LIN {X -19.393, Y 137.224, Z 298.25, A 0, B 90, C 0, E1 0, E2 0, E3 0, E4 0} C_DIS
LIN {X -14.94, Y 135.645, Z 298.25, A 0, B 90, C 0, E1 0, E2 0, E3 0, E4 0} C_DIS
LIN {X -10.792, Y 133.376, Z 298.25, A 0, B 90, C 0, E1 0, E2 0, E3 0, E4 0} C_DIS
LIN {X -6.941, Y 130.631, Z 298.25, A 0, B 90, C 0, E1 0, E2 0, E3 0, E4 0} C_DIS
LIN {X -3.341, Y 127.563, Z 298.25, A 0, B 90, C 0, E1 0, E2 0, E3 0, E4 0} C_DIS
LIN {X 0, Y 124.352, Z 298.25, A 0, B 90, C 0, E1 0, E2 0, E3 0, E4 0} C_DIS
LIN {X 3.004, Y 120.935, Z 298.25, A 0, B 90, C 0, E1 0, E2 0, E3 0, E4 0} C_DIS
LIN {X 6.227, Y 117.473, Z 298.25, A 0, B 90, C 0, E1 0, E2 0, E3 0, E4 0} C_DIS
LIN {X 9.503, Y 114.059, Z 298.25, A 0, B 90, C 0, E1 0, E2 0, E3 0, E4 0} C_DIS
LIN {X 12.968, Y 110.84, Z 298.25, A 0, B 90, C 0, E1 0, E2 0, E3 0, E4 0} C_DIS
LIN {X 16.832, Y 108.123, Z 298.25, A 0, B 90, C 0, E1 0, E2 0, E3 0, E4 0} C_DIS
LIN {X 21.253, Y 106.495, Z 298.25, A 0, B 90, C 0, E1 0, E2 0, E3 0, E4 0} C_DIS
LIN {X 25.964, Y 106.394, Z 298.25, A 0, B 90, C 0, E1 0, E2 0, E3 0, E4 0} C_DIS
LIN {X 30.572, Y 107.44, Z 298.25, A 0, B 90, C 0, E1 0, E2 0, E3 0, E4 0} C_DIS
LIN {X 35.02, Y 109.05, Z 298.25, A 0, B 90, C 0, E1 0, E2 0, E3 0, E4 0} C_DIS
LIN {X 39.382, Y 110.883, Z 298.25, A 0, B 90, C 0, E1 0, E2 0, E3 0, E4 0} C_DIS
LIN {X 43.728, Y 112.754, Z 298.25, A 0, B 90, C 0, E1 0, E2 0, E3 0, E4 0} C_DIS
LIN {X 48.108, Y 114.542, Z 298.25, A 0, B 90, C 0, E1 0, E2 0, E3 0, E4 0} C_DIS
LIN {X 52.558, Y 116.148, Z 298.25, A 0, B 90, C 0, E1 0, E2 0, E3 0, E4 0} C_DIS
LIN {X 57.101, Y 117.467, Z 298.25, A 0, B 90, C 0, E1 0, E2 0, E3 0, E4 0} C_DIS
LIN {X 61.743, Y 118.371, Z 298.25, A 0, B 90, C 0, E1 0, E2 0, E3 0, E4 0} C_DIS
LIN {X 66.459, Y 118.689, Z 298.25, A 0, B 90, C 0, E1 0, E2 0, E3 0, E4 0} C_DIS
LIN {X 71.159, Y 118.207, Z 298.25, A 0, B 90, C 0, E1 0, E2 0, E3 0, E4 0} C_DIS
LIN {X 75.634, Y 116.707, Z 298.25, A 0, B 90, C 0, E1 0, E2 0, E3 0, E4 0} C_DIS
LIN {X 79.57, Y 114.108, Z 298.25, A 0, B 90, C 0, E1 0, E2 0, E3 0, E4 0} C_DIS
LIN {X 82.708, Y 110.582, Z 298.25, A 0, B 90, C 0, E1 0, E2 0, E3 0, E4 0} C_DIS
LIN {X 84.997, Y 106.45, Z 298.25, A 0, B 90, C 0, E1 0, E2 0, E3 0, E4 0} C_DIS
LIN {X 86.553, Y 101.986, Z 298.25, A 0, B 90, C 0, E1 0, E2 0, E3 0, E4 0} C_DIS
LIN {X 87.536, Y 97.36, Z 298.25, A 0, B 90, C 0, E1 0, E2 0, E3 0, E4 0} C_DIS
LIN {X 88.091, Y 92.663, Z 298.25, A 0, B 90, C 0, E1 0, E2 0, E3 0, E4 0} C_DIS
LIN {X 88.341, Y 87.938, Z 298.25, A 0, B 90, C 0, E1 0, E2 0, E3 0, E4 0} C_DIS
LIN {X 88.398, Y 83.207, Z 298.25, A 0, B 90, C 0, E1 0, E2 0, E3 0, E4 0} C_DIS
LIN {X 88.377, Y 78.476, Z 298.25, A 0, B 90, C 0, E1 0, E2 0, E3 0, E4 0} C_DIS
LIN {X 88.427, Y 73.745, Z 298.25, A 0, B 90, C 0, E1 0, E2 0, E3 0, E4 0} C_DIS
LIN {X 88.78, Y 69.029, Z 298.25, A 0, B 90, C 0, E1 0, E2 0, E3 0, E4 0} C_DIS
LIN {X 89.835, Y 64.425, Z 298.25, A 0, B 90, C 0, E1 0, E2 0, E3 0, E4 0} C_DIS
LIN {X 92.094, Y 60.292, Z 298.25, A 0, B 90, C 0, E1 0, E2 0, E3 0, E4 0} C_DIS
LIN {X 95.553, Y 57.088, Z 298.25, A 0, B 90, C 0, E1 0, E2 0, E3 0, E4 0} C_DIS
LIN {X 99.64, Y 54.714, Z 298.25, A 0, B 90, C 0, E1 0, E2 0, E3 0, E4 0} C_DIS
LIN {X 103.963, Y 52.792, Z 298.25, A 0, B 90, C 0, E1 0, E2 0, E3 0, E4 0} C_DIS
LIN {X 108.359, Y 51.043, Z 298.25, A 0, B 90, C 0, E1 0, E2 0, E3 0, E4 0} C_DIS
LIN {X 112.757, Y 49.297, Z 298.25, A 0, B 90, C 0, E1 0, E2 0, E3 0, E4 0} C_DIS
LIN {X 117.106, Y 47.436, Z 298.25, A 0, B 90, C 0, E1 0, E2 0, E3 0, E4 0} C_DIS
LIN {X 121.359, Y 45.364, Z 298.25, A 0, B 90, C 0, E1 0, E2 0, E3 0, E4 0} C_DIS
LIN {X 125.45, Y 42.989, Z 298.25, A 0, B 90, C 0, E1 0, E2 0, E3 0, E4 0} C_DIS
LIN {X 129.281, Y 40.217, Z 298.25, A 0, B 90, C 0, E1 0, E2 0, E3 0, E4 0} C_DIS
LIN {X 132.696, Y 36.95, Z 298.25, A 0, B 90, C 0, E1 0, E2 0, E3 0, E4 0} C_DIS
LIN {X 135.457, Y 33.118, Z 298.25, A 0, B 90, C 0, E1 0, E2 0, E3 0, E4 0} C_DIS
LIN {X 137.252, Y 28.754, Z 298.25, A 0, B 90, C 0, E1 0, E2 0, E3 0, E4 0} C_DIS
LIN {X 137.838, Y 24.073, Z 298.25, A 0, B 90, C 0, E1 0, E2 0, E3 0, E4 0} C_DIS
LIN {X 137.224, Y 19.393, Z 298.25, A 0, B 90, C 0, E1 0, E2 0, E3 0, E4 0} C_DIS
LIN {X 135.645, Y 14.94, Z 298.25, A 0, B 90, C 0, E1 0, E2 0, E3 0, E4 0} C_DIS
LIN {X 133.376, Y 10.792, Z 298.25, A 0, B 90, C 0, E1 0, E2 0, E3 0, E4 0} C_DIS
LIN {X 130.631, Y 6.941, Z 298.25, A 0, B 90, C 0, E1 0, E2 0, E3 0, E4 0} C_DIS
LIN {X 127.563, Y 3.341, Z 298.25, A 0, B 90, C 0, E1 0, E2 0, E3 0, E4 0} C_DIS
LIN {X 124.352, Y 0, Z 298.25, A 0, B 90, C 0, E1 0, E2 0, E3 0, E4 0} C_DIS
LIN {X 120.935, Y -3.004, Z 298.25, A 0, B 90, C 0, E1 0, E2 0, E3 0, E4 0} C_DIS
LIN {X 117.473, Y -6.227, Z 298.25, A 0, B 90, C 0, E1 0, E2 0, E3 0, E4 0} C_DIS
LIN {X 114.059, Y -9.503, Z 298.25, A 0, B 90, C 0, E1 0, E2 0, E3 0, E4 0} C_DIS
LIN {X 110.84, Y -12.968, Z 298.25, A 0, B 90, C 0, E1 0, E2 0, E3 0, E4 0} C_DIS
LIN {X 108.123, Y -16.832, Z 298.25, A 0, B 90, C 0, E1 0, E2 0, E3 0, E4 0} C_DIS
LIN {X 106.495, Y -21.253, Z 298.25, A 0, B 90, C 0, E1 0, E2 0, E3 0, E4 0} C_DIS
LIN {X 106.394, Y -25.964, Z 298.25, A 0, B 90, C 0, E1 0, E2 0, E3 0, E4 0} C_DIS
LIN {X 107.44, Y -30.572, Z 298.25, A 0, B 90, C 0, E1 0, E2 0, E3 0, E4 0} C_DIS
LIN {X 109.05, Y -35.02, Z 298.25, A 0, B 90, C 0, E1 0, E2 0, E3 0, E4 0} C_DIS
LIN {X 110.883, Y -39.382, Z 298.25, A 0, B 90, C 0, E1 0, E2 0, E3 0, E4 0} C_DIS
LIN {X 112.754, Y -43.728, Z 298.25, A 0, B 90, C 0, E1 0, E2 0, E3 0, E4 0} C_DIS
LIN {X 114.542, Y -48.108, Z 298.25, A 0, B 90, C 0, E1 0, E2 0, E3 0, E4 0} C_DIS
LIN {X 116.148, Y -52.558, Z 298.25, A 0, B 90, C 0, E1 0, E2 0, E3 0, E4 0} C_DIS
LIN {X 117.467, Y -57.101, Z 298.25, A 0, B 90, C 0, E1 0, E2 0, E3 0, E4 0} C_DIS
LIN {X 118.371, Y -61.743, Z 298.25, A 0, B 90, C 0, E1 0, E2 0, E3 0, E4 0} C_DIS
LIN {X 118.689, Y -66.459, Z 298.25, A 0, B 90, C 0, E1 0, E2 0, E3 0, E4 0} C_DIS
LIN {X 118.207, Y -71.159, Z 298.25, A 0, B 90, C 0, E1 0, E2 0, E3 0, E4 0} C_DIS
LIN {X 116.707, Y -75.634, Z 298.25, A 0, B 90, C 0, E1 0, E2 0, E3 0, E4 0} C_DIS
LIN {X 114.108, Y -79.57, Z 298.25, A 0, B 90, C 0, E1 0, E2 0, E3 0, E4 0} C_DIS
LIN {X 110.582, Y -82.708, Z 298.25, A 0, B 90, C 0, E1 0, E2 0, E3 0, E4 0} C_DIS
LIN {X 106.45, Y -84.997, Z 298.25, A 0, B 90, C 0, E1 0, E2 0, E3 0, E4 0} C_DIS
LIN {X 101.986, Y -86.553, Z 298.25, A 0, B 90, C 0, E1 0, E2 0, E3 0, E4 0} C_DIS
LIN {X 97.36, Y -87.536, Z 298.25, A 0, B 90, C 0, E1 0, E2 0, E3 0, E4 0} C_DIS
LIN {X 92.663, Y -88.091, Z 298.25, A 0, B 90, C 0, E1 0, E2 0, E3 0, E4 0} C_DIS
LIN {X 87.938, Y -88.341, Z 298.25, A 0, B 90, C 0, E1 0, E2 0, E3 0, E4 0} C_DIS
LIN {X 83.207, Y -88.398, Z 298.25, A 0, B 90, C 0, E1 0, E2 0, E3 0, E4 0} C_DIS
LIN {X 78.476, Y -88.377, Z 298.25, A 0, B 90, C 0, E1 0, E2 0, E3 0, E4 0} C_DIS
LIN {X 73.745, Y -88.427, Z 298.25, A 0, B 90, C 0, E1 0, E2 0, E3 0, E4 0} C_DIS
LIN {X 69.029, Y -88.78, Z 298.25, A 0, B 90, C 0, E1 0, E2 0, E3 0, E4 0} C_DIS
LIN {X 64.425, Y -89.835, Z 298.25, A 0, B 90, C 0, E1 0, E2 0, E3 0, E4 0} C_DIS
LIN {X 60.292, Y -92.094, Z 298.25, A 0, B 90, C 0, E1 0, E2 0, E3 0, E4 0} C_DIS
LIN {X 57.088, Y -95.553, Z 298.25, A 0, B 90, C 0, E1 0, E2 0, E3 0, E4 0} C_DIS
LIN {X 54.714, Y -99.64, Z 298.25, A 0, B 90, C 0, E1 0, E2 0, E3 0, E4 0} C_DIS
LIN {X 52.792, Y -103.963, Z 298.25, A 0, B 90, C 0, E1 0, E2 0, E3 0, E4 0} C_DIS
LIN {X 51.043, Y -108.359, Z 298.25, A 0, B 90, C 0, E1 0, E2 0, E3 0, E4 0} C_DIS
LIN {X 49.297, Y -112.757, Z 298.25, A 0, B 90, C 0, E1 0, E2 0, E3 0, E4 0} C_DIS
LIN {X 47.436, Y -117.106, Z 298.25, A 0, B 90, C 0, E1 0, E2 0, E3 0, E4 0} C_DIS
LIN {X 45.364, Y -121.359, Z 298.25, A 0, B 90, C 0, E1 0, E2 0, E3 0, E4 0} C_DIS
LIN {X 42.989, Y -125.45, Z 298.25, A 0, B 90, C 0, E1 0, E2 0, E3 0, E4 0} C_DIS
LIN {X 40.217, Y -129.281, Z 298.25, A 0, B 90, C 0, E1 0, E2 0, E3 0, E4 0} C_DIS
LIN {X 36.95, Y -132.696, Z 298.25, A 0, B 90, C 0, E1 0, E2 0, E3 0, E4 0} C_DIS
LIN {X 33.118, Y -135.457, Z 298.25, A 0, B 90, C 0, E1 0, E2 0, E3 0, E4 0} C_DIS
LIN {X 28.754, Y -137.252, Z 298.25, A 0, B 90, C 0, E1 0, E2 0, E3 0, E4 0} C_DIS
LIN {X 24.073, Y -137.838, Z 298.25, A 0, B 90, C 0, E1 0, E2 0, E3 0, E4 0} C_DIS
LIN {X 19.393, Y -137.224, Z 298.25, A 0, B 90, C 0, E1 0, E2 0, E3 0, E4 0} C_DIS
LIN {X 14.94, Y -135.645, Z 298.25, A 0, B 90, C 0, E1 0, E2 0, E3 0, E4 0} C_DIS
LIN {X 10.792, Y -133.376, Z 298.25, A 0, B 90, C 0, E1 0, E2 0, E3 0, E4 0} C_DIS
LIN {X 6.941, Y -130.631, Z 298.25, A 0, B 90, C 0, E1 0, E2 0, E3 0, E4 0} C_DIS
LIN {X 3.341, Y -127.563, Z 298.25, A 0, B 90, C 0, E1 0, E2 0, E3 0, E4 0} C_DIS
LIN {X 0, Y -124.352, Z 298.25, A 0, B 90, C 0, E1 0, E2 0, E3 0, E4 0} C_DIS
LIN {X -3.004, Y -120.935, Z 298.25, A 0, B 90, C 0, E1 0, E2 0, E3 0, E4 0} C_DIS
LIN {X -6.227, Y -117.473, Z 298.25, A 0, B 90, C 0, E1 0, E2 0, E3 0, E4 0} C_DIS
LIN {X -9.503, Y -114.059, Z 298.25, A 0, B 90, C 0, E1 0, E2 0, E3 0, E4 0} C_DIS
LIN {X -12.968, Y -110.84, Z 298.25, A 0, B 90, C 0, E1 0, E2 0, E3 0, E4 0} C_DIS
LIN {X -16.832, Y -108.123, Z 298.25, A 0, B 90, C 0, E1 0, E2 0, E3 0, E4 0} C_DIS
LIN {X -21.253, Y -106.495, Z 298.25, A 0, B 90, C 0, E1 0, E2 0, E3 0, E4 0} C_DIS
LIN {X -25.964, Y -106.394, Z 298.25, A 0, B 90, C 0, E1 0, E2 0, E3 0, E4 0} C_DIS
LIN {X -30.572, Y -107.44, Z 298.25, A 0, B 90, C 0, E1 0, E2 0, E3 0, E4 0} C_DIS
LIN {X -35.02, Y -109.05, Z 298.25, A 0, B 90, C 0, E1 0, E2 0, E3 0, E4 0} C_DIS
LIN {X -39.382, Y -110.883, Z 298.25, A 0, B 90, C 0, E1 0, E2 0, E3 0, E4 0} C_DIS
LIN {X -43.728, Y -112.754, Z 298.25, A 0, B 90, C 0, E1 0, E2 0, E3 0, E4 0} C_DIS
LIN {X -48.108, Y -114.542, Z 298.25, A 0, B 90, C 0, E1 0, E2 0, E3 0, E4 0} C_DIS
LIN {X -52.558, Y -116.148, Z 298.25, A 0, B 90, C 0, E1 0, E2 0, E3 0, E4 0} C_DIS
LIN {X -57.101, Y -117.467, Z 298.25, A 0, B 90, C 0, E1 0, E2 0, E3 0, E4 0} C_DIS
LIN {X -61.743, Y -118.371, Z 298.25, A 0, B 90, C 0, E1 0, E2 0, E3 0, E4 0} C_DIS
LIN {X -66.459, Y -118.689, Z 298.25, A 0, B 90, C 0, E1 0, E2 0, E3 0, E4 0} C_DIS
LIN {X -71.159, Y -118.207, Z 298.25, A 0, B 90, C 0, E1 0, E2 0, E3 0, E4 0} C_DIS
LIN {X -75.634, Y -116.707, Z 298.25, A 0, B 90, C 0, E1 0, E2 0, E3 0, E4 0} C_DIS
LIN {X -79.57, Y -114.108, Z 298.25, A 0, B 90, C 0, E1 0, E2 0, E3 0, E4 0} C_DIS
LIN {X -82.708, Y -110.582, Z 298.25, A 0, B 90, C 0, E1 0, E2 0, E3 0, E4 0} C_DIS
LIN {X -84.997, Y -106.45, Z 298.25, A 0, B 90, C 0, E1 0, E2 0, E3 0, E4 0} C_DIS
LIN {X -86.553, Y -101.986, Z 298.25, A 0, B 90, C 0, E1 0, E2 0, E3 0, E4 0} C_DIS
LIN {X -87.536, Y -97.36, Z 298.25, A 0, B 90, C 0, E1 0, E2 0, E3 0, E4 0} C_DIS
LIN {X -88.091, Y -92.663, Z 298.25, A 0, B 90, C 0, E1 0, E2 0, E3 0, E4 0} C_DIS
LIN {X -88.341, Y -87.938, Z 298.25, A 0, B 90, C 0, E1 0, E2 0, E3 0, E4 0} C_DIS
LIN {X -88.398, Y -83.207, Z 298.25, A 0, B 90, C 0, E1 0, E2 0, E3 0, E4 0} C_DIS
LIN {X -88.377, Y -78.476, Z 298.25, A 0, B 90, C 0, E1 0, E2 0, E3 0, E4 0} C_DIS
LIN {X -88.427, Y -73.745, Z 298.25, A 0, B 90, C 0, E1 0, E2 0, E3 0, E4 0} C_DIS
LIN {X -88.78, Y -69.029, Z 298.25, A 0, B 90, C 0, E1 0, E2 0, E3 0, E4 0} C_DIS
LIN {X -89.835, Y -64.425, Z 298.25, A 0, B 90, C 0, E1 0, E2 0, E3 0, E4 0} C_DIS
LIN {X -92.094, Y -60.292, Z 298.25, A 0, B 90, C 0, E1 0, E2 0, E3 0, E4 0} C_DIS
LIN {X -95.553, Y -57.088, Z 298.25, A 0, B 90, C 0, E1 0, E2 0, E3 0, E4 0} C_DIS
LIN {X -99.64, Y -54.714, Z 298.25, A 0, B 90, C 0, E1 0, E2 0, E3 0, E4 0} C_DIS
LIN {X -103.963, Y -52.792, Z 298.25, A 0, B 90, C 0, E1 0, E2 0, E3 0, E4 0} C_DIS
LIN {X -108.359, Y -51.043, Z 298.25, A 0, B 90, C 0, E1 0, E2 0, E3 0, E4 0} C_DIS
LIN {X -112.757, Y -49.297, Z 298.25, A 0, B 90, C 0, E1 0, E2 0, E3 0, E4 0} C_DIS
LIN {X -117.106, Y -47.436, Z 298.25, A 0, B 90, C 0, E1 0, E2 0, E3 0, E4 0} C_DIS
LIN {X -121.359, Y -45.364, Z 298.25, A 0, B 90, C 0, E1 0, E2 0, E3 0, E4 0} C_DIS
LIN {X -125.45, Y -42.989, Z 298.25, A 0, B 90, C 0, E1 0, E2 0, E3 0, E4 0} C_DIS
LIN {X -129.281, Y -40.217, Z 298.25, A 0, B 90, C 0, E1 0, E2 0, E3 0, E4 0} C_DIS
LIN {X -132.696, Y -36.95, Z 298.25, A 0, B 90, C 0, E1 0, E2 0, E3 0, E4 0} C_DIS
LIN {X -135.457, Y -33.118, Z 298.25, A 0, B 90, C 0, E1 0, E2 0, E3 0, E4 0} C_DIS
LIN {X -137.252, Y -28.754, Z 298.25, A 0, B 90, C 0, E1 0, E2 0, E3 0, E4 0} C_DIS
LIN {X -137.838, Y -24.073, Z 298.25, A 0, B 90, C 0, E1 0, E2 0, E3 0, E4 0} C_DIS
LIN {X -137.224, Y -19.393, Z 298.25, A 0, B 90, C 0, E1 0, E2 0, E3 0, E4 0} C_DIS
LIN {X -135.645, Y -14.94, Z 298.25, A 0, B 90, C 0, E1 0, E2 0, E3 0, E4 0} C_DIS
LIN {X -133.376, Y -10.792, Z 298.25, A 0, B 90, C 0, E1 0, E2 0, E3 0, E4 0} C_DIS
LIN {X -130.631, Y -6.941, Z 298.25, A 0, B 90, C 0, E1 0, E2 0, E3 0, E4 0} C_DIS
LIN {X -127.563, Y -3.341, Z 298.25, A 0, B 90, C 0, E1 0, E2 0, E3 0, E4 0} C_DIS
LIN {X -125.319, Y 0, Z 300.75, A 0, B 90, C 0, E1 0, E2 0, E3 0, E4 0} C_DIS
LIN {X -121.855, Y 3.043, Z 300.75, A 0, B 90, C 0, E1 0, E2 0, E3 0, E4 0} C_DIS
LIN {X -118.342, Y 6.3, Z 300.75, A 0, B 90, C 0, E1 0, E2 0, E3 0, E4 0} C_DIS
LIN {X -114.881, Y 9.612, Z 300.75, A 0, B 90, C 0, E1 0, E2 0, E3 0, E4 0} C_DIS
LIN {X -111.625, Y 13.124, Z 300.75, A 0, B 90, C 0, E1 0, E2 0, E3 0, E4 0} C_DIS
LIN {X -108.897, Y 17.052, Z 300.75, A 0, B 90, C 0, E1 0, E2 0, E3 0, E4 0} C_DIS
LIN {X -107.308, Y 21.549, Z 300.75, A 0, B 90, C 0, E1 0, E2 0, E3 0, E4 0} C_DIS
LIN {X -107.291, Y 26.32, Z 300.75, A 0, B 90, C 0, E1 0, E2 0, E3 0, E4 0} C_DIS
LIN {X -108.43, Y 30.967, Z 300.75, A 0, B 90, C 0, E1 0, E2 0, E3 0, E4 0} C_DIS
LIN {X -110.13, Y 35.445, Z 300.75, A 0, B 90, C 0, E1 0, E2 0, E3 0, E4 0} C_DIS
LIN {X -112.047, Y 39.836, Z 300.75, A 0, B 90, C 0, E1 0, E2 0, E3 0, E4 0} C_DIS
LIN {X -113.995, Y 44.212, Z 300.75, A 0, B 90, C 0, E1 0, E2 0, E3 0, E4 0} C_DIS
LIN {X -115.852, Y 48.629, Z 300.75, A 0, B 90, C 0, E1 0, E2 0, E3 0, E4 0} C_DIS
LIN {X -117.516, Y 53.121, Z 300.75, A 0, B 90, C 0, E1 0, E2 0, E3 0, E4 0} C_DIS
LIN {X -118.876, Y 57.713, Z 300.75, A 0, B 90, C 0, E1 0, E2 0, E3 0, E4 0} C_DIS
LIN {X -119.801, Y 62.411, Z 300.75, A 0, B 90, C 0, E1 0, E2 0, E3 0, E4 0} C_DIS
LIN {X -120.113, Y 67.188, Z 300.75, A 0, B 90, C 0, E1 0, E2 0, E3 0, E4 0} C_DIS
LIN {X -119.591, Y 71.942, Z 300.75, A 0, B 90, C 0, E1 0, E2 0, E3 0, E4 0} C_DIS
LIN {X -118.014, Y 76.452, Z 300.75, A 0, B 90, C 0, E1 0, E2 0, E3 0, E4 0} C_DIS
LIN {X -115.31, Y 80.389, Z 300.75, A 0, B 90, C 0, E1 0, E2 0, E3 0, E4 0} C_DIS
LIN {X -111.675, Y 83.492, Z 300.75, A 0, B 90, C 0, E1 0, E2 0, E3 0, E4 0} C_DIS
LIN {X -107.444, Y 85.723, Z 300.75, A 0, B 90, C 0, E1 0, E2 0, E3 0, E4 0} C_DIS
LIN {X -102.895, Y 87.212, Z 300.75, A 0, B 90, C 0, E1 0, E2 0, E3 0, E4 0} C_DIS
LIN {X -98.194, Y 88.123, Z 300.75, A 0, B 90, C 0, E1 0, E2 0, E3 0, E4 0} C_DIS
LIN {X -93.428, Y 88.603, Z 300.75, A 0, B 90, C 0, E1 0, E2 0, E3 0, E4 0} C_DIS
LIN {X -88.641, Y 88.778, Z 300.75, A 0, B 90, C 0, E1 0, E2 0, E3 0, E4 0} C_DIS
LIN {X -83.851, Y 88.757, Z 300.75, A 0, B 90, C 0, E1 0, E2 0, E3 0, E4 0} C_DIS
LIN {X -79.061, Y 88.659, Z 300.75, A 0, B 90, C 0, E1 0, E2 0, E3 0, E4 0} C_DIS
LIN {X -74.27, Y 88.63, Z 300.75, A 0, B 90, C 0, E1 0, E2 0, E3 0, E4 0} C_DIS
LIN {X -69.489, Y 88.903, Z 300.75, A 0, B 90, C 0, E1 0, E2 0, E3 0, E4 0} C_DIS
LIN {X -64.808, Y 89.881, Z 300.75, A 0, B 90, C 0, E1 0, E2 0, E3 0, E4 0} C_DIS
LIN {X -60.582, Y 92.09, Z 300.75, A 0, B 90, C 0, E1 0, E2 0, E3 0, E4 0} C_DIS
LIN {X -57.303, Y 95.559, Z 300.75, A 0, B 90, C 0, E1 0, E2 0, E3 0, E4 0} C_DIS
LIN {X -54.9, Y 99.697, Z 300.75, A 0, B 90, C 0, E1 0, E2 0, E3 0, E4 0} C_DIS
LIN {X -52.978, Y 104.085, Z 300.75, A 0, B 90, C 0, E1 0, E2 0, E3 0, E4 0} C_DIS
LIN {X -51.248, Y 108.552, Z 300.75, A 0, B 90, C 0, E1 0, E2 0, E3 0, E4 0} C_DIS
LIN {X -49.53, Y 113.025, Z 300.75, A 0, B 90, C 0, E1 0, E2 0, E3 0, E4 0} C_DIS
LIN {X -47.703, Y 117.453, Z 300.75, A 0, B 90, C 0, E1 0, E2 0, E3 0, E4 0} C_DIS
LIN {X -45.666, Y 121.789, Z 300.75, A 0, B 90, C 0, E1 0, E2 0, E3 0, E4 0} C_DIS
LIN {X -43.327, Y 125.968, Z 300.75, A 0, B 90, C 0, E1 0, E2 0, E3 0, E4 0} C_DIS
LIN {X -40.587, Y 129.894, Z 300.75, A 0, B 90, C 0, E1 0, E2 0, E3 0, E4 0} C_DIS
LIN {X -37.343, Y 133.413, Z 300.75, A 0, B 90, C 0, E1 0, E2 0, E3 0, E4 0} C_DIS
LIN {X -33.518, Y 136.284, Z 300.75, A 0, B 90, C 0, E1 0, E2 0, E3 0, E4 0} C_DIS
LIN {X -29.136, Y 138.187, Z 300.75, A 0, B 90, C 0, E1 0, E2 0, E3 0, E4 0} C_DIS
LIN {X -24.407, Y 138.861, Z 300.75, A 0, B 90, C 0, E1 0, E2 0, E3 0, E4 0} C_DIS
LIN {X -19.661, Y 138.298, Z 300.75, A 0, B 90, C 0, E1 0, E2 0, E3 0, E4 0} C_DIS
LIN {X -15.141, Y 136.734, Z 300.75, A 0, B 90, C 0, E1 0, E2 0, E3 0, E4 0} C_DIS
LIN {X -10.932, Y 134.453, Z 300.75, A 0, B 90, C 0, E1 0, E2 0, E3 0, E4 0} C_DIS
LIN {X -7.028, Y 131.68, Z 300.75, A 0, B 90, C 0, E1 0, E2 0, E3 0, E4 0} C_DIS
LIN {X -3.382, Y 128.575, Z 300.75, A 0, B 90, C 0, E1 0, E2 0, E3 0, E4 0} C_DIS
LIN {X 0, Y 125.319, Z 300.75, A 0, B 90, C 0, E1 0, E2 0, E3 0, E4 0} C_DIS
LIN {X 3.043, Y 121.855, Z 300.75, A 0, B 90, C 0, E1 0, E2 0, E3 0, E4 0} C_DIS
LIN {X 6.3, Y 118.342, Z 300.75, A 0, B 90, C 0, E1 0, E2 0, E3 0, E4 0} C_DIS
LIN {X 9.612, Y 114.881, Z 300.75, A 0, B 90, C 0, E1 0, E2 0, E3 0, E4 0} C_DIS
LIN {X 13.124, Y 111.625, Z 300.75, A 0, B 90, C 0, E1 0, E2 0, E3 0, E4 0} C_DIS
LIN {X 17.052, Y 108.897, Z 300.75, A 0, B 90, C 0, E1 0, E2 0, E3 0, E4 0} C_DIS
LIN {X 21.549, Y 107.308, Z 300.75, A 0, B 90, C 0, E1 0, E2 0, E3 0, E4 0} C_DIS
LIN {X 26.32, Y 107.291, Z 300.75, A 0, B 90, C 0, E1 0, E2 0, E3 0, E4 0} C_DIS
LIN {X 30.967, Y 108.43, Z 300.75, A 0, B 90, C 0, E1 0, E2 0, E3 0, E4 0} C_DIS
LIN {X 35.445, Y 110.13, Z 300.75, A 0, B 90, C 0, E1 0, E2 0, E3 0, E4 0} C_DIS
LIN {X 39.836, Y 112.047, Z 300.75, A 0, B 90, C 0, E1 0, E2 0, E3 0, E4 0} C_DIS
LIN {X 44.212, Y 113.995, Z 300.75, A 0, B 90, C 0, E1 0, E2 0, E3 0, E4 0} C_DIS
LIN {X 48.629, Y 115.852, Z 300.75, A 0, B 90, C 0, E1 0, E2 0, E3 0, E4 0} C_DIS
LIN {X 53.121, Y 117.516, Z 300.75, A 0, B 90, C 0, E1 0, E2 0, E3 0, E4 0} C_DIS
LIN {X 57.713, Y 118.876, Z 300.75, A 0, B 90, C 0, E1 0, E2 0, E3 0, E4 0} C_DIS
LIN {X 62.411, Y 119.801, Z 300.75, A 0, B 90, C 0, E1 0, E2 0, E3 0, E4 0} C_DIS
LIN {X 67.188, Y 120.113, Z 300.75, A 0, B 90, C 0, E1 0, E2 0, E3 0, E4 0} C_DIS
LIN {X 71.942, Y 119.591, Z 300.75, A 0, B 90, C 0, E1 0, E2 0, E3 0, E4 0} C_DIS
LIN {X 76.452, Y 118.014, Z 300.75, A 0, B 90, C 0, E1 0, E2 0, E3 0, E4 0} C_DIS
LIN {X 80.389, Y 115.31, Z 300.75, A 0, B 90, C 0, E1 0, E2 0, E3 0, E4 0} C_DIS
LIN {X 83.492, Y 111.675, Z 300.75, A 0, B 90, C 0, E1 0, E2 0, E3 0, E4 0} C_DIS
LIN {X 85.723, Y 107.444, Z 300.75, A 0, B 90, C 0, E1 0, E2 0, E3 0, E4 0} C_DIS
LIN {X 87.212, Y 102.895, Z 300.75, A 0, B 90, C 0, E1 0, E2 0, E3 0, E4 0} C_DIS
LIN {X 88.123, Y 98.194, Z 300.75, A 0, B 90, C 0, E1 0, E2 0, E3 0, E4 0} C_DIS
LIN {X 88.603, Y 93.428, Z 300.75, A 0, B 90, C 0, E1 0, E2 0, E3 0, E4 0} C_DIS
LIN {X 88.778, Y 88.641, Z 300.75, A 0, B 90, C 0, E1 0, E2 0, E3 0, E4 0} C_DIS
LIN {X 88.757, Y 83.851, Z 300.75, A 0, B 90, C 0, E1 0, E2 0, E3 0, E4 0} C_DIS
LIN {X 88.659, Y 79.061, Z 300.75, A 0, B 90, C 0, E1 0, E2 0, E3 0, E4 0} C_DIS
LIN {X 88.63, Y 74.27, Z 300.75, A 0, B 90, C 0, E1 0, E2 0, E3 0, E4 0} C_DIS
LIN {X 88.903, Y 69.489, Z 300.75, A 0, B 90, C 0, E1 0, E2 0, E3 0, E4 0} C_DIS
LIN {X 89.881, Y 64.808, Z 300.75, A 0, B 90, C 0, E1 0, E2 0, E3 0, E4 0} C_DIS
LIN {X 92.09, Y 60.582, Z 300.75, A 0, B 90, C 0, E1 0, E2 0, E3 0, E4 0} C_DIS
LIN {X 95.559, Y 57.303, Z 300.75, A 0, B 90, C 0, E1 0, E2 0, E3 0, E4 0} C_DIS
LIN {X 99.697, Y 54.9, Z 300.75, A 0, B 90, C 0, E1 0, E2 0, E3 0, E4 0} C_DIS
LIN {X 104.085, Y 52.978, Z 300.75, A 0, B 90, C 0, E1 0, E2 0, E3 0, E4 0} C_DIS
LIN {X 108.552, Y 51.248, Z 300.75, A 0, B 90, C 0, E1 0, E2 0, E3 0, E4 0} C_DIS
LIN {X 113.025, Y 49.53, Z 300.75, A 0, B 90, C 0, E1 0, E2 0, E3 0, E4 0} C_DIS
LIN {X 117.453, Y 47.703, Z 300.75, A 0, B 90, C 0, E1 0, E2 0, E3 0, E4 0} C_DIS
LIN {X 121.789, Y 45.666, Z 300.75, A 0, B 90, C 0, E1 0, E2 0, E3 0, E4 0} C_DIS
LIN {X 125.968, Y 43.327, Z 300.75, A 0, B 90, C 0, E1 0, E2 0, E3 0, E4 0} C_DIS
LIN {X 129.894, Y 40.587, Z 300.75, A 0, B 90, C 0, E1 0, E2 0, E3 0, E4 0} C_DIS
LIN {X 133.413, Y 37.343, Z 300.75, A 0, B 90, C 0, E1 0, E2 0, E3 0, E4 0} C_DIS
LIN {X 136.284, Y 33.518, Z 300.75, A 0, B 90, C 0, E1 0, E2 0, E3 0, E4 0} C_DIS
LIN {X 138.187, Y 29.136, Z 300.75, A 0, B 90, C 0, E1 0, E2 0, E3 0, E4 0} C_DIS
LIN {X 138.861, Y 24.407, Z 300.75, A 0, B 90, C 0, E1 0, E2 0, E3 0, E4 0} C_DIS
LIN {X 138.298, Y 19.661, Z 300.75, A 0, B 90, C 0, E1 0, E2 0, E3 0, E4 0} C_DIS
LIN {X 136.734, Y 15.141, Z 300.75, A 0, B 90, C 0, E1 0, E2 0, E3 0, E4 0} C_DIS
LIN {X 134.453, Y 10.932, Z 300.75, A 0, B 90, C 0, E1 0, E2 0, E3 0, E4 0} C_DIS
LIN {X 131.68, Y 7.028, Z 300.75, A 0, B 90, C 0, E1 0, E2 0, E3 0, E4 0} C_DIS
LIN {X 128.575, Y 3.382, Z 300.75, A 0, B 90, C 0, E1 0, E2 0, E3 0, E4 0} C_DIS
LIN {X 125.319, Y 0, Z 300.75, A 0, B 90, C 0, E1 0, E2 0, E3 0, E4 0} C_DIS
LIN {X 121.855, Y -3.043, Z 300.75, A 0, B 90, C 0, E1 0, E2 0, E3 0, E4 0} C_DIS
LIN {X 118.342, Y -6.3, Z 300.75, A 0, B 90, C 0, E1 0, E2 0, E3 0, E4 0} C_DIS
LIN {X 114.881, Y -9.612, Z 300.75, A 0, B 90, C 0, E1 0, E2 0, E3 0, E4 0} C_DIS
LIN {X 111.625, Y -13.124, Z 300.75, A 0, B 90, C 0, E1 0, E2 0, E3 0, E4 0} C_DIS
LIN {X 108.897, Y -17.052, Z 300.75, A 0, B 90, C 0, E1 0, E2 0, E3 0, E4 0} C_DIS
LIN {X 107.308, Y -21.549, Z 300.75, A 0, B 90, C 0, E1 0, E2 0, E3 0, E4 0} C_DIS
LIN {X 107.291, Y -26.32, Z 300.75, A 0, B 90, C 0, E1 0, E2 0, E3 0, E4 0} C_DIS
LIN {X 108.43, Y -30.967, Z 300.75, A 0, B 90, C 0, E1 0, E2 0, E3 0, E4 0} C_DIS
LIN {X 110.13, Y -35.445, Z 300.75, A 0, B 90, C 0, E1 0, E2 0, E3 0, E4 0} C_DIS
LIN {X 112.047, Y -39.836, Z 300.75, A 0, B 90, C 0, E1 0, E2 0, E3 0, E4 0} C_DIS
LIN {X 113.995, Y -44.212, Z 300.75, A 0, B 90, C 0, E1 0, E2 0, E3 0, E4 0} C_DIS
LIN {X 115.852, Y -48.629, Z 300.75, A 0, B 90, C 0, E1 0, E2 0, E3 0, E4 0} C_DIS
LIN {X 117.516, Y -53.121, Z 300.75, A 0, B 90, C 0, E1 0, E2 0, E3 0, E4 0} C_DIS
LIN {X 118.876, Y -57.713, Z 300.75, A 0, B 90, C 0, E1 0, E2 0, E3 0, E4 0} C_DIS
LIN {X 119.801, Y -62.411, Z 300.75, A 0, B 90, C 0, E1 0, E2 0, E3 0, E4 0} C_DIS
LIN {X 120.113, Y -67.188, Z 300.75, A 0, B 90, C 0, E1 0, E2 0, E3 0, E4 0} C_DIS
LIN {X 119.591, Y -71.942, Z 300.75, A 0, B 90, C 0, E1 0, E2 0, E3 0, E4 0} C_DIS
LIN {X 118.014, Y -76.452, Z 300.75, A 0, B 90, C 0, E1 0, E2 0, E3 0, E4 0} C_DIS
LIN {X 115.31, Y -80.389, Z 300.75, A 0, B 90, C 0, E1 0, E2 0, E3 0, E4 0} C_DIS
LIN {X 111.675, Y -83.492, Z 300.75, A 0, B 90, C 0, E1 0, E2 0, E3 0, E4 0} C_DIS
LIN {X 107.444, Y -85.723, Z 300.75, A 0, B 90, C 0, E1 0, E2 0, E3 0, E4 0} C_DIS
LIN {X 102.895, Y -87.212, Z 300.75, A 0, B 90, C 0, E1 0, E2 0, E3 0, E4 0} C_DIS
LIN {X 98.194, Y -88.123, Z 300.75, A 0, B 90, C 0, E1 0, E2 0, E3 0, E4 0} C_DIS
LIN {X 93.428, Y -88.603, Z 300.75, A 0, B 90, C 0, E1 0, E2 0, E3 0, E4 0} C_DIS
LIN {X 88.641, Y -88.778, Z 300.75, A 0, B 90, C 0, E1 0, E2 0, E3 0, E4 0} C_DIS
LIN {X 83.851, Y -88.757, Z 300.75, A 0, B 90, C 0, E1 0, E2 0, E3 0, E4 0} C_DIS
LIN {X 79.061, Y -88.659, Z 300.75, A 0, B 90, C 0, E1 0, E2 0, E3 0, E4 0} C_DIS
LIN {X 74.27, Y -88.63, Z 300.75, A 0, B 90, C 0, E1 0, E2 0, E3 0, E4 0} C_DIS
LIN {X 69.489, Y -88.903, Z 300.75, A 0, B 90, C 0, E1 0, E2 0, E3 0, E4 0} C_DIS
LIN {X 64.808, Y -89.881, Z 300.75, A 0, B 90, C 0, E1 0, E2 0, E3 0, E4 0} C_DIS
LIN {X 60.582, Y -92.09, Z 300.75, A 0, B 90, C 0, E1 0, E2 0, E3 0, E4 0} C_DIS
LIN {X 57.303, Y -95.559, Z 300.75, A 0, B 90, C 0, E1 0, E2 0, E3 0, E4 0} C_DIS
LIN {X 54.9, Y -99.697, Z 300.75, A 0, B 90, C 0, E1 0, E2 0, E3 0, E4 0} C_DIS
LIN {X 52.978, Y -104.085, Z 300.75, A 0, B 90, C 0, E1 0, E2 0, E3 0, E4 0} C_DIS
LIN {X 51.248, Y -108.552, Z 300.75, A 0, B 90, C 0, E1 0, E2 0, E3 0, E4 0} C_DIS
LIN {X 49.53, Y -113.025, Z 300.75, A 0, B 90, C 0, E1 0, E2 0, E3 0, E4 0} C_DIS
LIN {X 47.703, Y -117.453, Z 300.75, A 0, B 90, C 0, E1 0, E2 0, E3 0, E4 0} C_DIS
LIN {X 45.666, Y -121.789, Z 300.75, A 0, B 90, C 0, E1 0, E2 0, E3 0, E4 0} C_DIS
LIN {X 43.327, Y -125.968, Z 300.75, A 0, B 90, C 0, E1 0, E2 0, E3 0, E4 0} C_DIS
LIN {X 40.587, Y -129.894, Z 300.75, A 0, B 90, C 0, E1 0, E2 0, E3 0, E4 0} C_DIS
LIN {X 37.343, Y -133.413, Z 300.75, A 0, B 90, C 0, E1 0, E2 0, E3 0, E4 0} C_DIS
LIN {X 33.518, Y -136.284, Z 300.75, A 0, B 90, C 0, E1 0, E2 0, E3 0, E4 0} C_DIS
LIN {X 29.136, Y -138.187, Z 300.75, A 0, B 90, C 0, E1 0, E2 0, E3 0, E4 0} C_DIS
LIN {X 24.407, Y -138.861, Z 300.75, A 0, B 90, C 0, E1 0, E2 0, E3 0, E4 0} C_DIS
LIN {X 19.661, Y -138.298, Z 300.75, A 0, B 90, C 0, E1 0, E2 0, E3 0, E4 0} C_DIS
LIN {X 15.141, Y -136.734, Z 300.75, A 0, B 90, C 0, E1 0, E2 0, E3 0, E4 0} C_DIS
LIN {X 10.932, Y -134.453, Z 300.75, A 0, B 90, C 0, E1 0, E2 0, E3 0, E4 0} C_DIS
LIN {X 7.028, Y -131.68, Z 300.75, A 0, B 90, C 0, E1 0, E2 0, E3 0, E4 0} C_DIS
LIN {X 3.382, Y -128.575, Z 300.75, A 0, B 90, C 0, E1 0, E2 0, E3 0, E4 0} C_DIS
LIN {X 0, Y -125.319, Z 300.75, A 0, B 90, C 0, E1 0, E2 0, E3 0, E4 0} C_DIS
LIN {X -3.043, Y -121.855, Z 300.75, A 0, B 90, C 0, E1 0, E2 0, E3 0, E4 0} C_DIS
LIN {X -6.3, Y -118.342, Z 300.75, A 0, B 90, C 0, E1 0, E2 0, E3 0, E4 0} C_DIS
LIN {X -9.612, Y -114.881, Z 300.75, A 0, B 90, C 0, E1 0, E2 0, E3 0, E4 0} C_DIS
LIN {X -13.124, Y -111.625, Z 300.75, A 0, B 90, C 0, E1 0, E2 0, E3 0, E4 0} C_DIS
LIN {X -17.052, Y -108.897, Z 300.75, A 0, B 90, C 0, E1 0, E2 0, E3 0, E4 0} C_DIS
LIN {X -21.549, Y -107.308, Z 300.75, A 0, B 90, C 0, E1 0, E2 0, E3 0, E4 0} C_DIS
LIN {X -26.32, Y -107.291, Z 300.75, A 0, B 90, C 0, E1 0, E2 0, E3 0, E4 0} C_DIS
LIN {X -30.967, Y -108.43, Z 300.75, A 0, B 90, C 0, E1 0, E2 0, E3 0, E4 0} C_DIS
LIN {X -35.445, Y -110.13, Z 300.75, A 0, B 90, C 0, E1 0, E2 0, E3 0, E4 0} C_DIS
LIN {X -39.836, Y -112.047, Z 300.75, A 0, B 90, C 0, E1 0, E2 0, E3 0, E4 0} C_DIS
LIN {X -44.212, Y -113.995, Z 300.75, A 0, B 90, C 0, E1 0, E2 0, E3 0, E4 0} C_DIS
LIN {X -48.629, Y -115.852, Z 300.75, A 0, B 90, C 0, E1 0, E2 0, E3 0, E4 0} C_DIS
LIN {X -53.121, Y -117.516, Z 300.75, A 0, B 90, C 0, E1 0, E2 0, E3 0, E4 0} C_DIS
LIN {X -57.713, Y -118.876, Z 300.75, A 0, B 90, C 0, E1 0, E2 0, E3 0, E4 0} C_DIS
LIN {X -62.411, Y -119.801, Z 300.75, A 0, B 90, C 0, E1 0, E2 0, E3 0, E4 0} C_DIS
LIN {X -67.188, Y -120.113, Z 300.75, A 0, B 90, C 0, E1 0, E2 0, E3 0, E4 0} C_DIS
LIN {X -71.942, Y -119.591, Z 300.75, A 0, B 90, C 0, E1 0, E2 0, E3 0, E4 0} C_DIS
LIN {X -76.452, Y -118.014, Z 300.75, A 0, B 90, C 0, E1 0, E2 0, E3 0, E4 0} C_DIS
LIN {X -80.389, Y -115.31, Z 300.75, A 0, B 90, C 0, E1 0, E2 0, E3 0, E4 0} C_DIS
LIN {X -83.492, Y -111.675, Z 300.75, A 0, B 90, C 0, E1 0, E2 0, E3 0, E4 0} C_DIS
LIN {X -85.723, Y -107.444, Z 300.75, A 0, B 90, C 0, E1 0, E2 0, E3 0, E4 0} C_DIS
LIN {X -87.212, Y -102.895, Z 300.75, A 0, B 90, C 0, E1 0, E2 0, E3 0, E4 0} C_DIS
LIN {X -88.123, Y -98.194, Z 300.75, A 0, B 90, C 0, E1 0, E2 0, E3 0, E4 0} C_DIS
LIN {X -88.603, Y -93.428, Z 300.75, A 0, B 90, C 0, E1 0, E2 0, E3 0, E4 0} C_DIS
LIN {X -88.778, Y -88.641, Z 300.75, A 0, B 90, C 0, E1 0, E2 0, E3 0, E4 0} C_DIS
LIN {X -88.757, Y -83.851, Z 300.75, A 0, B 90, C 0, E1 0, E2 0, E3 0, E4 0} C_DIS
LIN {X -88.659, Y -79.061, Z 300.75, A 0, B 90, C 0, E1 0, E2 0, E3 0, E4 0} C_DIS
LIN {X -88.63, Y -74.27, Z 300.75, A 0, B 90, C 0, E1 0, E2 0, E3 0, E4 0} C_DIS
LIN {X -88.903, Y -69.489, Z 300.75, A 0, B 90, C 0, E1 0, E2 0, E3 0, E4 0} C_DIS
LIN {X -89.881, Y -64.808, Z 300.75, A 0, B 90, C 0, E1 0, E2 0, E3 0, E4 0} C_DIS
LIN {X -92.09, Y -60.582, Z 300.75, A 0, B 90, C 0, E1 0, E2 0, E3 0, E4 0} C_DIS
LIN {X -95.559, Y -57.303, Z 300.75, A 0, B 90, C 0, E1 0, E2 0, E3 0, E4 0} C_DIS
LIN {X -99.697, Y -54.9, Z 300.75, A 0, B 90, C 0, E1 0, E2 0, E3 0, E4 0} C_DIS
LIN {X -104.085, Y -52.978, Z 300.75, A 0, B 90, C 0, E1 0, E2 0, E3 0, E4 0} C_DIS
LIN {X -108.552, Y -51.248, Z 300.75, A 0, B 90, C 0, E1 0, E2 0, E3 0, E4 0} C_DIS
LIN {X -113.025, Y -49.53, Z 300.75, A 0, B 90, C 0, E1 0, E2 0, E3 0, E4 0} C_DIS
LIN {X -117.453, Y -47.703, Z 300.75, A 0, B 90, C 0, E1 0, E2 0, E3 0, E4 0} C_DIS
LIN {X -121.789, Y -45.666, Z 300.75, A 0, B 90, C 0, E1 0, E2 0, E3 0, E4 0} C_DIS
LIN {X -125.968, Y -43.327, Z 300.75, A 0, B 90, C 0, E1 0, E2 0, E3 0, E4 0} C_DIS
LIN {X -129.894, Y -40.587, Z 300.75, A 0, B 90, C 0, E1 0, E2 0, E3 0, E4 0} C_DIS
LIN {X -133.413, Y -37.343, Z 300.75, A 0, B 90, C 0, E1 0, E2 0, E3 0, E4 0} C_DIS
LIN {X -136.284, Y -33.518, Z 300.75, A 0, B 90, C 0, E1 0, E2 0, E3 0, E4 0} C_DIS
LIN {X -138.187, Y -29.136, Z 300.75, A 0, B 90, C 0, E1 0, E2 0, E3 0, E4 0} C_DIS
LIN {X -138.861, Y -24.407, Z 300.75, A 0, B 90, C 0, E1 0, E2 0, E3 0, E4 0} C_DIS
LIN {X -138.298, Y -19.661, Z 300.75, A 0, B 90, C 0, E1 0, E2 0, E3 0, E4 0} C_DIS
LIN {X -136.734, Y -15.141, Z 300.75, A 0, B 90, C 0, E1 0, E2 0, E3 0, E4 0} C_DIS
LIN {X -134.453, Y -10.932, Z 300.75, A 0, B 90, C 0, E1 0, E2 0, E3 0, E4 0} C_DIS
LIN {X -131.68, Y -7.028, Z 300.75, A 0, B 90, C 0, E1 0, E2 0, E3 0, E4 0} C_DIS
LIN {X -128.575, Y -3.382, Z 300.75, A 0, B 90, C 0, E1 0, E2 0, E3 0, E4 0} C_DIS
LIN {X -126.297, Y 0, Z 303.25, A 0, B 90, C 0, E1 0, E2 0, E3 0, E4 0} C_DIS
LIN {X -122.783, Y 3.083, Z 303.25, A 0, B 90, C 0, E1 0, E2 0, E3 0, E4 0} C_DIS
LIN {X -119.219, Y 6.373, Z 303.25, A 0, B 90, C 0, E1 0, E2 0, E3 0, E4 0} C_DIS
LIN {X -115.711, Y 9.723, Z 303.25, A 0, B 90, C 0, E1 0, E2 0, E3 0, E4 0} C_DIS
LIN {X -112.418, Y 13.283, Z 303.25, A 0, B 90, C 0, E1 0, E2 0, E3 0, E4 0} C_DIS
LIN {X -109.679, Y 17.277, Z 303.25, A 0, B 90, C 0, E1 0, E2 0, E3 0, E4 0} C_DIS
LIN {X -108.132, Y 21.85, Z 303.25, A 0, B 90, C 0, E1 0, E2 0, E3 0, E4 0} C_DIS
LIN {X -108.2, Y 26.681, Z 303.25, A 0, B 90, C 0, E1 0, E2 0, E3 0, E4 0} C_DIS
LIN {X -109.433, Y 31.367, Z 303.25, A 0, B 90, C 0, E1 0, E2 0, E3 0, E4 0} C_DIS
LIN {X -111.222, Y 35.875, Z 303.25, A 0, B 90, C 0, E1 0, E2 0, E3 0, E4 0} C_DIS
LIN {X -113.223, Y 40.293, Z 303.25, A 0, B 90, C 0, E1 0, E2 0, E3 0, E4 0} C_DIS
LIN {X -115.25, Y 44.701, Z 303.25, A 0, B 90, C 0, E1 0, E2 0, E3 0, E4 0} C_DIS
LIN {X -117.176, Y 49.153, Z 303.25, A 0, B 90, C 0, E1 0, E2 0, E3 0, E4 0} C_DIS
LIN {X -118.896, Y 53.689, Z 303.25, A 0, B 90, C 0, E1 0, E2 0, E3 0, E4 0} C_DIS
LIN {X -120.298, Y 58.332, Z 303.25, A 0, B 90, C 0, E1 0, E2 0, E3 0, E4 0} C_DIS
LIN {X -121.244, Y 63.087, Z 303.25, A 0, B 90, C 0, E1 0, E2 0, E3 0, E4 0} C_DIS
LIN {X -121.549, Y 67.924, Z 303.25, A 0, B 90, C 0, E1 0, E2 0, E3 0, E4 0} C_DIS
LIN {X -120.984, Y 72.733, Z 303.25, A 0, B 90, C 0, E1 0, E2 0, E3 0, E4 0} C_DIS
LIN {X -119.326, Y 77.278, Z 303.25, A 0, B 90, C 0, E1 0, E2 0, E3 0, E4 0} C_DIS
LIN {X -116.515, Y 81.213, Z 303.25, A 0, B 90, C 0, E1 0, E2 0, E3 0, E4 0} C_DIS
LIN {X -112.771, Y 84.279, Z 303.25, A 0, B 90, C 0, E1 0, E2 0, E3 0, E4 0} C_DIS
LIN {X -108.442, Y 86.452, Z 303.25, A 0, B 90, C 0, E1 0, E2 0, E3 0, E4 0} C_DIS
LIN {X -103.808, Y 87.872, Z 303.25, A 0, B 90, C 0, E1 0, E2 0, E3 0, E4 0} C_DIS
LIN {X -99.032, Y 88.711, Z 303.25, A 0, B 90, C 0, E1 0, E2 0, E3 0, E4 0} C_DIS
LIN {X -94.199, Y 89.117, Z 303.25, A 0, B 90, C 0, E1 0, E2 0, E3 0, E4 0} C_DIS
LIN {X -89.349, Y 89.217, Z 303.25, A 0, B 90, C 0, E1 0, E2 0, E3 0, E4 0} C_DIS
LIN {X -84.499, Y 89.12, Z 303.25, A 0, B 90, C 0, E1 0, E2 0, E3 0, E4 0} C_DIS
LIN {X -79.651, Y 88.944, Z 303.25, A 0, B 90, C 0, E1 0, E2 0, E3 0, E4 0} C_DIS
LIN {X -74.801, Y 88.837, Z 303.25, A 0, B 90, C 0, E1 0, E2 0, E3 0, E4 0} C_DIS
LIN {X -69.956, Y 89.03, Z 303.25, A 0, B 90, C 0, E1 0, E2 0, E3 0, E4 0} C_DIS
LIN {X -65.197, Y 89.928, Z 303.25, A 0, B 90, C 0, E1 0, E2 0, E3 0, E4 0} C_DIS
LIN {X -60.877, Y 92.085, Z 303.25, A 0, B 90, C 0, E1 0, E2 0, E3 0, E4 0} C_DIS
LIN {X -57.522, Y 95.561, Z 303.25, A 0, B 90, C 0, E1 0, E2 0, E3 0, E4 0} C_DIS
LIN {X -55.086, Y 99.75, Z 303.25, A 0, B 90, C 0, E1 0, E2 0, E3 0, E4 0} C_DIS
LIN {X -53.164, Y 104.203, Z 303.25, A 0, B 90, C 0, E1 0, E2 0, E3 0, E4 0} C_DIS
LIN {X -51.452, Y 108.742, Z 303.25, A 0, B 90, C 0, E1 0, E2 0, E3 0, E4 0} C_DIS
LIN {X -49.762, Y 113.289, Z 303.25, A 0, B 90, C 0, E1 0, E2 0, E3 0, E4 0} C_DIS
LIN {X -47.968, Y 117.796, Z 303.25, A 0, B 90, C 0, E1 0, E2 0, E3 0, E4 0} C_DIS
LIN {X -45.968, Y 122.215, Z 303.25, A 0, B 90, C 0, E1 0, E2 0, E3 0, E4 0} C_DIS
LIN {X -43.665, Y 126.483, Z 303.25, A 0, B 90, C 0, E1 0, E2 0, E3 0, E4 0} C_DIS
LIN {X -40.957, Y 130.505, Z 303.25, A 0, B 90, C 0, E1 0, E2 0, E3 0, E4 0} C_DIS
LIN {X -37.738, Y 134.128, Z 303.25, A 0, B 90, C 0, E1 0, E2 0, E3 0, E4 0} C_DIS
LIN {X -33.922, Y 137.11, Z 303.25, A 0, B 90, C 0, E1 0, E2 0, E3 0, E4 0} C_DIS
LIN {X -29.524, Y 139.124, Z 303.25, A 0, B 90, C 0, E1 0, E2 0, E3 0, E4 0} C_DIS
LIN {X -24.749, Y 139.888, Z 303.25, A 0, B 90, C 0, E1 0, E2 0, E3 0, E4 0} C_DIS
LIN {X -19.936, Y 139.379, Z 303.25, A 0, B 90, C 0, E1 0, E2 0, E3 0, E4 0} C_DIS
LIN {X -15.347, Y 137.832, Z 303.25, A 0, B 90, C 0, E1 0, E2 0, E3 0, E4 0} C_DIS
LIN {X -11.075, Y 135.541, Z 303.25, A 0, B 90, C 0, E1 0, E2 0, E3 0, E4 0} C_DIS
LIN {X -7.117, Y 132.74, Z 303.25, A 0, B 90, C 0, E1 0, E2 0, E3 0, E4 0} C_DIS
LIN {X -3.423, Y 129.598, Z 303.25, A 0, B 90, C 0, E1 0, E2 0, E3 0, E4 0} C_DIS
LIN {X 0, Y 126.297, Z 303.25, A 0, B 90, C 0, E1 0, E2 0, E3 0, E4 0} C_DIS
LIN {X 3.083, Y 122.783, Z 303.25, A 0, B 90, C 0, E1 0, E2 0, E3 0, E4 0} C_DIS
LIN {X 6.373, Y 119.219, Z 303.25, A 0, B 90, C 0, E1 0, E2 0, E3 0, E4 0} C_DIS
LIN {X 9.723, Y 115.711, Z 303.25, A 0, B 90, C 0, E1 0, E2 0, E3 0, E4 0} C_DIS
LIN {X 13.283, Y 112.418, Z 303.25, A 0, B 90, C 0, E1 0, E2 0, E3 0, E4 0} C_DIS
LIN {X 17.277, Y 109.679, Z 303.25, A 0, B 90, C 0, E1 0, E2 0, E3 0, E4 0} C_DIS
LIN {X 21.85, Y 108.132, Z 303.25, A 0, B 90, C 0, E1 0, E2 0, E3 0, E4 0} C_DIS
LIN {X 26.681, Y 108.2, Z 303.25, A 0, B 90, C 0, E1 0, E2 0, E3 0, E4 0} C_DIS
LIN {X 31.367, Y 109.433, Z 303.25, A 0, B 90, C 0, E1 0, E2 0, E3 0, E4 0} C_DIS
LIN {X 35.875, Y 111.222, Z 303.25, A 0, B 90, C 0, E1 0, E2 0, E3 0, E4 0} C_DIS
LIN {X 40.293, Y 113.223, Z 303.25, A 0, B 90, C 0, E1 0, E2 0, E3 0, E4 0} C_DIS
LIN {X 44.701, Y 115.25, Z 303.25, A 0, B 90, C 0, E1 0, E2 0, E3 0, E4 0} C_DIS
LIN {X 49.153, Y 117.176, Z 303.25, A 0, B 90, C 0, E1 0, E2 0, E3 0, E4 0} C_DIS
LIN {X 53.689, Y 118.896, Z 303.25, A 0, B 90, C 0, E1 0, E2 0, E3 0, E4 0} C_DIS
LIN {X 58.332, Y 120.298, Z 303.25, A 0, B 90, C 0, E1 0, E2 0, E3 0, E4 0} C_DIS
LIN {X 63.087, Y 121.244, Z 303.25, A 0, B 90, C 0, E1 0, E2 0, E3 0, E4 0} C_DIS
LIN {X 67.924, Y 121.549, Z 303.25, A 0, B 90, C 0, E1 0, E2 0, E3 0, E4 0} C_DIS
LIN {X 72.733, Y 120.984, Z 303.25, A 0, B 90, C 0, E1 0, E2 0, E3 0, E4 0} C_DIS
LIN {X 77.278, Y 119.326, Z 303.25, A 0, B 90, C 0, E1 0, E2 0, E3 0, E4 0} C_DIS
LIN {X 81.213, Y 116.515, Z 303.25, A 0, B 90, C 0, E1 0, E2 0, E3 0, E4 0} C_DIS
LIN {X 84.279, Y 112.771, Z 303.25, A 0, B 90, C 0, E1 0, E2 0, E3 0, E4 0} C_DIS
LIN {X 86.452, Y 108.442, Z 303.25, A 0, B 90, C 0, E1 0, E2 0, E3 0, E4 0} C_DIS
LIN {X 87.872, Y 103.808, Z 303.25, A 0, B 90, C 0, E1 0, E2 0, E3 0, E4 0} C_DIS
LIN {X 88.711, Y 99.032, Z 303.25, A 0, B 90, C 0, E1 0, E2 0, E3 0, E4 0} C_DIS
LIN {X 89.117, Y 94.199, Z 303.25, A 0, B 90, C 0, E1 0, E2 0, E3 0, E4 0} C_DIS
LIN {X 89.217, Y 89.349, Z 303.25, A 0, B 90, C 0, E1 0, E2 0, E3 0, E4 0} C_DIS
LIN {X 89.12, Y 84.499, Z 303.25, A 0, B 90, C 0, E1 0, E2 0, E3 0, E4 0} C_DIS
LIN {X 88.944, Y 79.651, Z 303.25, A 0, B 90, C 0, E1 0, E2 0, E3 0, E4 0} C_DIS
LIN {X 88.837, Y 74.801, Z 303.25, A 0, B 90, C 0, E1 0, E2 0, E3 0, E4 0} C_DIS
LIN {X 89.03, Y 69.956, Z 303.25, A 0, B 90, C 0, E1 0, E2 0, E3 0, E4 0} C_DIS
LIN {X 89.928, Y 65.197, Z 303.25, A 0, B 90, C 0, E1 0, E2 0, E3 0, E4 0} C_DIS
LIN {X 92.085, Y 60.877, Z 303.25, A 0, B 90, C 0, E1 0, E2 0, E3 0, E4 0} C_DIS
LIN {X 95.561, Y 57.522, Z 303.25, A 0, B 90, C 0, E1 0, E2 0, E3 0, E4 0} C_DIS
LIN {X 99.75, Y 55.086, Z 303.25, A 0, B 90, C 0, E1 0, E2 0, E3 0, E4 0} C_DIS
LIN {X 104.203, Y 53.164, Z 303.25, A 0, B 90, C 0, E1 0, E2 0, E3 0, E4 0} C_DIS
LIN {X 108.742, Y 51.452, Z 303.25, A 0, B 90, C 0, E1 0, E2 0, E3 0, E4 0} C_DIS
LIN {X 113.289, Y 49.762, Z 303.25, A 0, B 90, C 0, E1 0, E2 0, E3 0, E4 0} C_DIS
LIN {X 117.796, Y 47.968, Z 303.25, A 0, B 90, C 0, E1 0, E2 0, E3 0, E4 0} C_DIS
LIN {X 122.215, Y 45.968, Z 303.25, A 0, B 90, C 0, E1 0, E2 0, E3 0, E4 0} C_DIS
LIN {X 126.483, Y 43.665, Z 303.25, A 0, B 90, C 0, E1 0, E2 0, E3 0, E4 0} C_DIS
LIN {X 130.505, Y 40.957, Z 303.25, A 0, B 90, C 0, E1 0, E2 0, E3 0, E4 0} C_DIS
LIN {X 134.128, Y 37.738, Z 303.25, A 0, B 90, C 0, E1 0, E2 0, E3 0, E4 0} C_DIS
LIN {X 137.11, Y 33.922, Z 303.25, A 0, B 90, C 0, E1 0, E2 0, E3 0, E4 0} C_DIS
LIN {X 139.124, Y 29.524, Z 303.25, A 0, B 90, C 0, E1 0, E2 0, E3 0, E4 0} C_DIS
LIN {X 139.888, Y 24.749, Z 303.25, A 0, B 90, C 0, E1 0, E2 0, E3 0, E4 0} C_DIS
LIN {X 139.379, Y 19.936, Z 303.25, A 0, B 90, C 0, E1 0, E2 0, E3 0, E4 0} C_DIS
LIN {X 137.832, Y 15.347, Z 303.25, A 0, B 90, C 0, E1 0, E2 0, E3 0, E4 0} C_DIS
LIN {X 135.541, Y 11.075, Z 303.25, A 0, B 90, C 0, E1 0, E2 0, E3 0, E4 0} C_DIS
LIN {X 132.74, Y 7.117, Z 303.25, A 0, B 90, C 0, E1 0, E2 0, E3 0, E4 0} C_DIS
LIN {X 129.598, Y 3.423, Z 303.25, A 0, B 90, C 0, E1 0, E2 0, E3 0, E4 0} C_DIS
LIN {X 126.297, Y 0, Z 303.25, A 0, B 90, C 0, E1 0, E2 0, E3 0, E4 0} C_DIS
LIN {X 122.783, Y -3.083, Z 303.25, A 0, B 90, C 0, E1 0, E2 0, E3 0, E4 0} C_DIS
LIN {X 119.219, Y -6.373, Z 303.25, A 0, B 90, C 0, E1 0, E2 0, E3 0, E4 0} C_DIS
LIN {X 115.711, Y -9.723, Z 303.25, A 0, B 90, C 0, E1 0, E2 0, E3 0, E4 0} C_DIS
LIN {X 112.418, Y -13.283, Z 303.25, A 0, B 90, C 0, E1 0, E2 0, E3 0, E4 0} C_DIS
LIN {X 109.679, Y -17.277, Z 303.25, A 0, B 90, C 0, E1 0, E2 0, E3 0, E4 0} C_DIS
LIN {X 108.132, Y -21.85, Z 303.25, A 0, B 90, C 0, E1 0, E2 0, E3 0, E4 0} C_DIS
LIN {X 108.2, Y -26.681, Z 303.25, A 0, B 90, C 0, E1 0, E2 0, E3 0, E4 0} C_DIS
LIN {X 109.433, Y -31.367, Z 303.25, A 0, B 90, C 0, E1 0, E2 0, E3 0, E4 0} C_DIS
LIN {X 111.222, Y -35.875, Z 303.25, A 0, B 90, C 0, E1 0, E2 0, E3 0, E4 0} C_DIS
LIN {X 113.223, Y -40.293, Z 303.25, A 0, B 90, C 0, E1 0, E2 0, E3 0, E4 0} C_DIS
LIN {X 115.25, Y -44.701, Z 303.25, A 0, B 90, C 0, E1 0, E2 0, E3 0, E4 0} C_DIS
LIN {X 117.176, Y -49.153, Z 303.25, A 0, B 90, C 0, E1 0, E2 0, E3 0, E4 0} C_DIS
LIN {X 118.896, Y -53.689, Z 303.25, A 0, B 90, C 0, E1 0, E2 0, E3 0, E4 0} C_DIS
LIN {X 120.298, Y -58.332, Z 303.25, A 0, B 90, C 0, E1 0, E2 0, E3 0, E4 0} C_DIS
LIN {X 121.244, Y -63.087, Z 303.25, A 0, B 90, C 0, E1 0, E2 0, E3 0, E4 0} C_DIS
LIN {X 121.549, Y -67.924, Z 303.25, A 0, B 90, C 0, E1 0, E2 0, E3 0, E4 0} C_DIS
LIN {X 120.984, Y -72.733, Z 303.25, A 0, B 90, C 0, E1 0, E2 0, E3 0, E4 0} C_DIS
LIN {X 119.326, Y -77.278, Z 303.25, A 0, B 90, C 0, E1 0, E2 0, E3 0, E4 0} C_DIS
LIN {X 116.515, Y -81.213, Z 303.25, A 0, B 90, C 0, E1 0, E2 0, E3 0, E4 0} C_DIS
LIN {X 112.771, Y -84.279, Z 303.25, A 0, B 90, C 0, E1 0, E2 0, E3 0, E4 0} C_DIS
LIN {X 108.442, Y -86.452, Z 303.25, A 0, B 90, C 0, E1 0, E2 0, E3 0, E4 0} C_DIS
LIN {X 103.808, Y -87.872, Z 303.25, A 0, B 90, C 0, E1 0, E2 0, E3 0, E4 0} C_DIS
LIN {X 99.032, Y -88.711, Z 303.25, A 0, B 90, C 0, E1 0, E2 0, E3 0, E4 0} C_DIS
LIN {X 94.199, Y -89.117, Z 303.25, A 0, B 90, C 0, E1 0, E2 0, E3 0, E4 0} C_DIS
LIN {X 89.349, Y -89.217, Z 303.25, A 0, B 90, C 0, E1 0, E2 0, E3 0, E4 0} C_DIS
LIN {X 84.499, Y -89.12, Z 303.25, A 0, B 90, C 0, E1 0, E2 0, E3 0, E4 0} C_DIS
LIN {X 79.651, Y -88.944, Z 303.25, A 0, B 90, C 0, E1 0, E2 0, E3 0, E4 0} C_DIS
LIN {X 74.801, Y -88.837, Z 303.25, A 0, B 90, C 0, E1 0, E2 0, E3 0, E4 0} C_DIS
LIN {X 69.956, Y -89.03, Z 303.25, A 0, B 90, C 0, E1 0, E2 0, E3 0, E4 0} C_DIS
LIN {X 65.197, Y -89.928, Z 303.25, A 0, B 90, C 0, E1 0, E2 0, E3 0, E4 0} C_DIS
LIN {X 60.877, Y -92.085, Z 303.25, A 0, B 90, C 0, E1 0, E2 0, E3 0, E4 0} C_DIS
LIN {X 57.522, Y -95.561, Z 303.25, A 0, B 90, C 0, E1 0, E2 0, E3 0, E4 0} C_DIS
LIN {X 55.086, Y -99.75, Z 303.25, A 0, B 90, C 0, E1 0, E2 0, E3 0, E4 0} C_DIS
LIN {X 53.164, Y -104.203, Z 303.25, A 0, B 90, C 0, E1 0, E2 0, E3 0, E4 0} C_DIS
LIN {X 51.452, Y -108.742, Z 303.25, A 0, B 90, C 0, E1 0, E2 0, E3 0, E4 0} C_DIS
LIN {X 49.762, Y -113.289, Z 303.25, A 0, B 90, C 0, E1 0, E2 0, E3 0, E4 0} C_DIS
LIN {X 47.968, Y -117.796, Z 303.25, A 0, B 90, C 0, E1 0, E2 0, E3 0, E4 0} C_DIS
LIN {X 45.968, Y -122.215, Z 303.25, A 0, B 90, C 0, E1 0, E2 0, E3 0, E4 0} C_DIS
LIN {X 43.665, Y -126.483, Z 303.25, A 0, B 90, C 0, E1 0, E2 0, E3 0, E4 0} C_DIS
LIN {X 40.957, Y -130.505, Z 303.25, A 0, B 90, C 0, E1 0, E2 0, E3 0, E4 0} C_DIS
LIN {X 37.738, Y -134.128, Z 303.25, A 0, B 90, C 0, E1 0, E2 0, E3 0, E4 0} C_DIS
LIN {X 33.922, Y -137.11, Z 303.25, A 0, B 90, C 0, E1 0, E2 0, E3 0, E4 0} C_DIS
LIN {X 29.524, Y -139.124, Z 303.25, A 0, B 90, C 0, E1 0, E2 0, E3 0, E4 0} C_DIS
LIN {X 24.749, Y -139.888, Z 303.25, A 0, B 90, C 0, E1 0, E2 0, E3 0, E4 0} C_DIS
LIN {X 19.936, Y -139.379, Z 303.25, A 0, B 90, C 0, E1 0, E2 0, E3 0, E4 0} C_DIS
LIN {X 15.347, Y -137.832, Z 303.25, A 0, B 90, C 0, E1 0, E2 0, E3 0, E4 0} C_DIS
LIN {X 11.075, Y -135.541, Z 303.25, A 0, B 90, C 0, E1 0, E2 0, E3 0, E4 0} C_DIS
LIN {X 7.117, Y -132.74, Z 303.25, A 0, B 90, C 0, E1 0, E2 0, E3 0, E4 0} C_DIS
LIN {X 3.423, Y -129.598, Z 303.25, A 0, B 90, C 0, E1 0, E2 0, E3 0, E4 0} C_DIS
LIN {X 0, Y -126.297, Z 303.25, A 0, B 90, C 0, E1 0, E2 0, E3 0, E4 0} C_DIS
LIN {X -3.083, Y -122.783, Z 303.25, A 0, B 90, C 0, E1 0, E2 0, E3 0, E4 0} C_DIS
LIN {X -6.373, Y -119.219, Z 303.25, A 0, B 90, C 0, E1 0, E2 0, E3 0, E4 0} C_DIS
LIN {X -9.723, Y -115.711, Z 303.25, A 0, B 90, C 0, E1 0, E2 0, E3 0, E4 0} C_DIS
LIN {X -13.283, Y -112.418, Z 303.25, A 0, B 90, C 0, E1 0, E2 0, E3 0, E4 0} C_DIS
LIN {X -17.277, Y -109.679, Z 303.25, A 0, B 90, C 0, E1 0, E2 0, E3 0, E4 0} C_DIS
LIN {X -21.85, Y -108.132, Z 303.25, A 0, B 90, C 0, E1 0, E2 0, E3 0, E4 0} C_DIS
LIN {X -26.681, Y -108.2, Z 303.25, A 0, B 90, C 0, E1 0, E2 0, E3 0, E4 0} C_DIS
LIN {X -31.367, Y -109.433, Z 303.25, A 0, B 90, C 0, E1 0, E2 0, E3 0, E4 0} C_DIS
LIN {X -35.875, Y -111.222, Z 303.25, A 0, B 90, C 0, E1 0, E2 0, E3 0, E4 0} C_DIS
LIN {X -40.293, Y -113.223, Z 303.25, A 0, B 90, C 0, E1 0, E2 0, E3 0, E4 0} C_DIS
LIN {X -44.701, Y -115.25, Z 303.25, A 0, B 90, C 0, E1 0, E2 0, E3 0, E4 0} C_DIS
LIN {X -49.153, Y -117.176, Z 303.25, A 0, B 90, C 0, E1 0, E2 0, E3 0, E4 0} C_DIS
LIN {X -53.689, Y -118.896, Z 303.25, A 0, B 90, C 0, E1 0, E2 0, E3 0, E4 0} C_DIS
LIN {X -58.332, Y -120.298, Z 303.25, A 0, B 90, C 0, E1 0, E2 0, E3 0, E4 0} C_DIS
LIN {X -63.087, Y -121.244, Z 303.25, A 0, B 90, C 0, E1 0, E2 0, E3 0, E4 0} C_DIS
LIN {X -67.924, Y -121.549, Z 303.25, A 0, B 90, C 0, E1 0, E2 0, E3 0, E4 0} C_DIS
LIN {X -72.733, Y -120.984, Z 303.25, A 0, B 90, C 0, E1 0, E2 0, E3 0, E4 0} C_DIS
LIN {X -77.278, Y -119.326, Z 303.25, A 0, B 90, C 0, E1 0, E2 0, E3 0, E4 0} C_DIS
LIN {X -81.213, Y -116.515, Z 303.25, A 0, B 90, C 0, E1 0, E2 0, E3 0, E4 0} C_DIS
LIN {X -84.279, Y -112.771, Z 303.25, A 0, B 90, C 0, E1 0, E2 0, E3 0, E4 0} C_DIS
LIN {X -86.452, Y -108.442, Z 303.25, A 0, B 90, C 0, E1 0, E2 0, E3 0, E4 0} C_DIS
LIN {X -87.872, Y -103.808, Z 303.25, A 0, B 90, C 0, E1 0, E2 0, E3 0, E4 0} C_DIS
LIN {X -88.711, Y -99.032, Z 303.25, A 0, B 90, C 0, E1 0, E2 0, E3 0, E4 0} C_DIS
LIN {X -89.117, Y -94.199, Z 303.25, A 0, B 90, C 0, E1 0, E2 0, E3 0, E4 0} C_DIS
LIN {X -89.217, Y -89.349, Z 303.25, A 0, B 90, C 0, E1 0, E2 0, E3 0, E4 0} C_DIS
LIN {X -89.12, Y -84.499, Z 303.25, A 0, B 90, C 0, E1 0, E2 0, E3 0, E4 0} C_DIS
LIN {X -88.944, Y -79.651, Z 303.25, A 0, B 90, C 0, E1 0, E2 0, E3 0, E4 0} C_DIS
LIN {X -88.837, Y -74.801, Z 303.25, A 0, B 90, C 0, E1 0, E2 0, E3 0, E4 0} C_DIS
LIN {X -89.03, Y -69.956, Z 303.25, A 0, B 90, C 0, E1 0, E2 0, E3 0, E4 0} C_DIS
LIN {X -89.928, Y -65.197, Z 303.25, A 0, B 90, C 0, E1 0, E2 0, E3 0, E4 0} C_DIS
LIN {X -92.085, Y -60.877, Z 303.25, A 0, B 90, C 0, E1 0, E2 0, E3 0, E4 0} C_DIS
LIN {X -95.561, Y -57.522, Z 303.25, A 0, B 90, C 0, E1 0, E2 0, E3 0, E4 0} C_DIS
LIN {X -99.75, Y -55.086, Z 303.25, A 0, B 90, C 0, E1 0, E2 0, E3 0, E4 0} C_DIS
LIN {X -104.203, Y -53.164, Z 303.25, A 0, B 90, C 0, E1 0, E2 0, E3 0, E4 0} C_DIS
LIN {X -108.742, Y -51.452, Z 303.25, A 0, B 90, C 0, E1 0, E2 0, E3 0, E4 0} C_DIS
LIN {X -113.289, Y -49.762, Z 303.25, A 0, B 90, C 0, E1 0, E2 0, E3 0, E4 0} C_DIS
LIN {X -117.796, Y -47.968, Z 303.25, A 0, B 90, C 0, E1 0, E2 0, E3 0, E4 0} C_DIS
LIN {X -122.215, Y -45.968, Z 303.25, A 0, B 90, C 0, E1 0, E2 0, E3 0, E4 0} C_DIS
LIN {X -126.483, Y -43.665, Z 303.25, A 0, B 90, C 0, E1 0, E2 0, E3 0, E4 0} C_DIS
LIN {X -130.505, Y -40.957, Z 303.25, A 0, B 90, C 0, E1 0, E2 0, E3 0, E4 0} C_DIS
LIN {X -134.128, Y -37.738, Z 303.25, A 0, B 90, C 0, E1 0, E2 0, E3 0, E4 0} C_DIS
LIN {X -137.11, Y -33.922, Z 303.25, A 0, B 90, C 0, E1 0, E2 0, E3 0, E4 0} C_DIS
LIN {X -139.124, Y -29.524, Z 303.25, A 0, B 90, C 0, E1 0, E2 0, E3 0, E4 0} C_DIS
LIN {X -139.888, Y -24.749, Z 303.25, A 0, B 90, C 0, E1 0, E2 0, E3 0, E4 0} C_DIS
LIN {X -139.379, Y -19.936, Z 303.25, A 0, B 90, C 0, E1 0, E2 0, E3 0, E4 0} C_DIS
LIN {X -137.832, Y -15.347, Z 303.25, A 0, B 90, C 0, E1 0, E2 0, E3 0, E4 0} C_DIS
LIN {X -135.541, Y -11.075, Z 303.25, A 0, B 90, C 0, E1 0, E2 0, E3 0, E4 0} C_DIS
LIN {X -132.74, Y -7.117, Z 303.25, A 0, B 90, C 0, E1 0, E2 0, E3 0, E4 0} C_DIS
LIN {X -129.598, Y -3.423, Z 303.25, A 0, B 90, C 0, E1 0, E2 0, E3 0, E4 0} C_DIS
LIN {X -129.598, Y -3.423, Z 453.25, A 0, B 90, C 0, E1 0, E2 0, E3 0, E4 0} C_DIS
PTP {A1 5, A2 -90, A3 100, A4 5, A5 -10, A6 90, E1 0, E2 0, E3 0, E4 0} C_PTP
;ENDFOLD

END
